FUNCTION_BLOCK FB_MotorSchuif IMPLEMENTS ITF_MotorSchuif				//MOTOR DIE KARTEN VAN DE PALLET NAAR DE ZIJKANT VERPLAATST
VAR_INPUT
END_VAR
VAR_OUTPUT
END_VAR
VAR
	
	StatusMotorSchuif : E_MotorSchuifStatus := E_MotorSchuifStatus.Kort;	//drie variabelen die worden gebruikt in de methods
	timerKort : TON;
	ErrorTrigger : BOOL; 
	
END_VAR

PROPERTY Status : E_MotorSchuifStatus
GET
Status := StatusMotorSchuif;
END_GET
SET
END_SET
END_PROPERTY

METHOD SturingKort : BOOL		//METHOD DIE DE SCHUIF INGETROKKEN ZET, DE SCHUIF HANGT NA DEZE METHOD RECHT BOVEN DE PALLET EN DUS KARTON
VAR_INPUT
END_VAR
IF ErrorTrigger THEN																//Controle error, ivm prioriteit bovenaan
    StatusMotorSchuif := E_MotorSchuifStatus.Error;
    SturingKort := FALSE;
    RETURN;
END_IF

IF StatusMotorSchuif <> E_MotorSchuifStatus.GoToKort AND							//Controle of sturing kort niet al eerder is geweest
   StatusMotorSchuif <> E_MotorSchuifStatus.Kort THEN	
   StatusMotorSchuif := E_MotorSchuifStatus.GoToKort;
    timerKort(IN := TRUE, PT := T#5S);
END_IF

IF StatusMotorSchuif = E_MotorSchuifStatus.GoToKort THEN							//Als het de eerste sturing kort is (GoToKort), wordt deze 5 seconde aangehouden en dan status kort
    timerKort(IN := TRUE, PT := T#5S);

    IF timerKort.Q THEN
        StatusMotorSchuif := E_MotorSchuifStatus.Kort;
		timerKort(IN := FALSE);
    END_IF
END_IF

SturingKort := TRUE;
END_METHOD

METHOD SturingLang : BOOL			//METHOD DIE DE SCHUIF UITGEDUWD ZET DUS KARTON HANGT NA DEZE STURING NAAST DE DEPALLETIZER
VAR_INPUT
END_VAR
IF ErrorTrigger THEN																//Controle error, ivm prioriteit bovenaan
    StatusMotorSchuif := E_MotorSchuifStatus.Error;
    SturingLang := FALSE;
    RETURN;
END_IF

IF StatusMotorSchuif <> E_MotorSchuifStatus.GoToLang AND							//Controle of sturing kort niet al eerder is geweest
   StatusMotorSchuif <> E_MotorSchuifStatus.Lang THEN
   StatusMotorSchuif := E_MotorSchuifStatus.GoToLang;
    timerKort(IN := TRUE, PT := T#5S);
END_IF

IF StatusMotorSchuif = E_MotorSchuifStatus.GoToLang THEN							//Als het de eerste sturing lang is (GoToLang), wordt deze 5 seconde aangehouden en dan status lang
    timerKort(IN := TRUE, PT := T#5S);

    IF timerKort.Q THEN
        StatusMotorSchuif := E_MotorSchuifStatus.Lang;
		timerKort(IN := FALSE);
    END_IF
END_IF

SturingLang := TRUE;
END_METHOD

END_FUNCTION_BLOCK

(* stored: Version 1.1.0.1
   POU FB_Motorschuif: Id {60d4b4a8-a1bb-4ed3-8c87-635035a0da9e}, SpecialFunc None
   Folder Methods: Id {cffb7d77-b82a-4ba3-8693-3a66c9404830}
   Folder Properties: Id {2bd36a5f-fa8f-4d44-809c-ed24ca09c9a3}
   Property Status: Id {30c9f538-9a28-4c6a-8549-dc11f43c5f81}
   Get Get: Id {8dfe6f5e-a6cb-4425-bc50-248ce4416186}
   Set Set: Id {4ddf90c4-c882-4ef3-b0ef-7d1663c4c9a4}
   Method SturingKort: Id {d310948d-e4e9-441e-8c2c-6b103810cceb}
   Method SturingLang: Id {54a6e14a-19cb-459d-8878-faf7b3492a1a} *)
